FUNCTION_BLOCK Controller
  (* Standard: 61499-2 *)
  (* Version 0,1, 2015-00-16, Th?o, PC_THEO *)
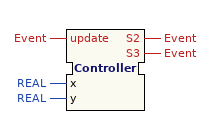
  EVENT_INPUT
    update;
  END_EVENT
  EVENT_OUTPUT
    S2;
    S3;
  END_EVENT
  VAR_INPUT
    x : REAL;
    y : REAL;
  END_VAR
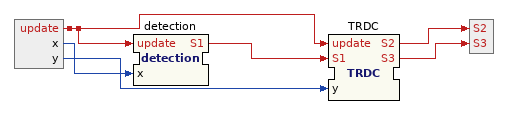
  FBS
    detection : detection;
    TRDC : TRDC;
  END_FBS
  EVENT_CONNECTIONS
    update TO detection.update;
    update TO TRDC.update;
    TRDC.S2 TO S2;
    TRDC.S3 TO S3;
    detection.S1 TO TRDC.S1;
  END_CONNECTIONS
  DATA_CONNECTIONS
    x TO detection.x;
    y TO TRDC.y;
  END_CONNECTIONS
END_FUNCTION_BLOCK
